// Mitsubishi GX Works2 project: 탈수기능 제어회로   PLC: Q02/Q02H

PROGRAM MAIN
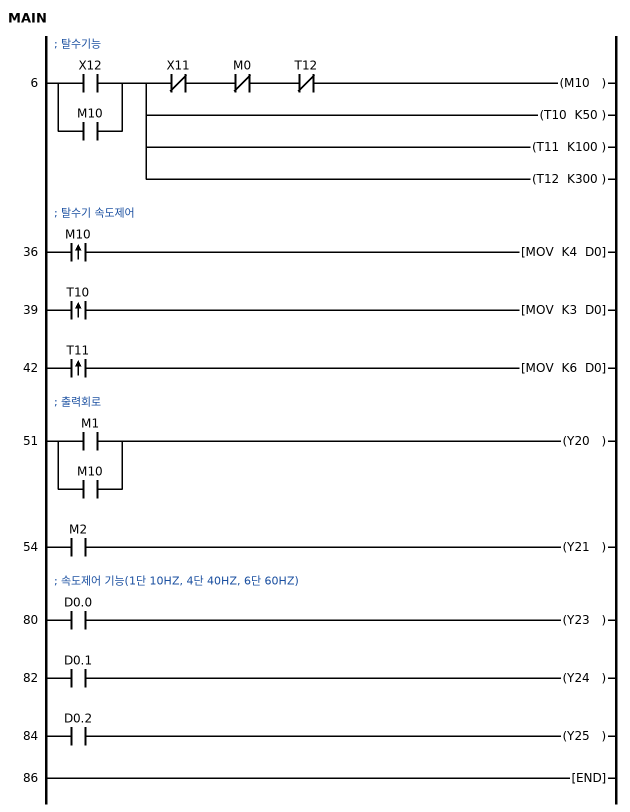
; 탈수기능
6     LD      X12
      OR      M10
      MPS
      ANI     X11
      ANI     M0
      ANI     T12
      OUT     M10
      MPP
      OUT     T10 K50
      OUT     T11 K100
      OUT     T12 K300
; 탈수기 속도제어
36    LDP     M10
      MOV     K4 D0
39    LDP     T10
      MOV     K3 D0
42    LDP     T11
      MOV     K6 D0
; 출력회로
51    LD      M1
      OR      M10
      OUT     Y20
54    LD      M2
      OUT     Y21
; 속도제어 기능(1단 10HZ, 4단 40HZ, 6단 60HZ)
80    LD      D0.0
      OUT     Y23
82    LD      D0.1
      OUT     Y24
84    LD      D0.2
      OUT     Y25
86    END
END_PROGRAM
